// TwinCAT 3 PLC project Sample01
// ProgramVersion: 3.1.4022.3
// libraries:
//   Tc2_Standard, * (Beckhoff Automation GmbH)
//   Tc2_System, * (Beckhoff Automation GmbH)
//   Tc3_Module, * (Beckhoff Automation GmbH)
// project tree:
//   DUTs/ E_States.TcDUT
//   / PlcTask.TcTTO
//   POUs/ FB_Machine.TcPOU, MAIN.TcPOU
// real-time tasks:
//   TASK PlcTask: cycle T#10ms, priority 20, ADS port 350

CONFIGURATION Sample01
    RESOURCE PLC ON TwinCAT3
        TASK PlcTask(INTERVAL := T#10ms, PRIORITY := 20);
        PROGRAM MAIN WITH PlcTask : MAIN;
    END_RESOURCE
END_CONFIGURATION

// ---- DUTs/E_States.TcDUT
{attribute 'qualified_only'}
{attribute 'strict'}
TYPE E_States :
(
	eWaiting := 0,
	eHasCoin,
	eProductEjected,
	eCoinEjected
);
END_TYPE

// ---- POUs/MAIN.TcPOU
PROGRAM MAIN
VAR
	fbMachine			:	FB_Machine(3);
	bButton				:	BOOL;
	bInsertCoin			:	BOOL;
	bTakeProduct		:	BOOL;
	bTakeCoin			:	BOOL;
END_VAR

fbMachine(	bButton	:= bButton,
			bInsertCoin := bInsertCoin,
			bTakeProduct := bTakeProduct,
			bTakeCoin := bTakeCoin);	

bButton := FALSE;
bInsertCoin := FALSE;
bTakeProduct := FALSE;
bTakeCoin := FALSE;

END_PROGRAM

// ---- POUs/FB_Machine.TcPOU
FUNCTION_BLOCK PUBLIC FB_Machine
VAR_INPUT
	bButton				:	BOOL;
	bInsertCoin			:	BOOL;
	bTakeProduct		:	BOOL;
	bTakeCoin			:	BOOL;	
END_VAR
VAR_OUTPUT
	eState 				:	E_States;
	nProducts			:	UINT;	
END_VAR
VAR
	rtrigButton			:	R_TRIG;
	rtrigInsertCoin		:	R_TRIG;
	rtrigTakeProduct	:	R_TRIG;
	rtrigTakeCoin		:	R_TRIG;
END_VAR

rtrigButton(CLK := bButton);
rtrigInsertCoin(CLK := bInsertCoin);
rtrigTakeProduct(CLK := bTakeProduct);
rtrigTakeCoin(CLK := bTakeCoin);

CASE eState OF
	E_States.eWaiting:
		IF (rtrigButton.Q) THEN
			;	// keep in the state
		END_IF
		IF (rtrigInsertCoin.Q) THEN
			ADSLOGSTR(msgCtrlMask := ADSLOG_MSGTYPE_HINT, msgFmtStr := 'Customer has insert a coin.', strArg := '');
			eState := E_States.eHasCoin;			
		END_IF
	E_States.eHasCoin:
		IF (rtrigButton.Q) THEN
			IF (nProducts > 0) THEN
				nProducts := nProducts - 1;
				ADSLOGSTR(msgCtrlMask := ADSLOG_MSGTYPE_HINT, msgFmtStr := 'Customer has pressed the button. Output product.', strArg := '');
				eState := E_States.eProductEjected;
			ELSE				
				ADSLOGSTR(msgCtrlMask := ADSLOG_MSGTYPE_HINT, msgFmtStr := 'Customer has pressed the button. No more products. Return coin.', strArg := '');
				eState := E_States.eCoinEjected;
			END_IF
		END_IF
	E_States.eProductEjected:
		IF (rtrigTakeProduct.Q) THEN
			ADSLOGSTR(msgCtrlMask := ADSLOG_MSGTYPE_HINT, msgFmtStr := 'Customer has taken the product.', strArg := '');
			eState := E_States.eWaiting;
		END_IF
	E_States.eCoinEjected:
		IF (rtrigTakeCoin.Q) THEN
			ADSLOGSTR(msgCtrlMask := ADSLOG_MSGTYPE_HINT, msgFmtStr := 'Customer has taken the coin.', strArg := '');
			eState := E_States.eWaiting;
		END_IF
	ELSE
		ADSLOGSTR(msgCtrlMask := ADSLOG_MSGTYPE_ERROR, msgFmtStr := 'Invalid state', strArg := '');
		eState := E_States.eWaiting;				
END_CASE

METHOD FB_init : BOOL
VAR_INPUT
	bInitRetains : BOOL; // if TRUE, the retain variables are initialized (warm start / cold start)
	bInCopyCode : BOOL;  // if TRUE, the instance afterwards gets moved into the copy code (online change)
	nProducts :	UINT;	
END_VAR
THIS^.nProducts := nProducts;
END_METHOD

END_FUNCTION_BLOCK
